// Writes an int64 field value, without a tag, to the stream.
FUNCTION F_WriteInt64 : HRESULT
VAR_INPUT
    stBuffer    : ST_Span;
END_VAR
VAR_IN_OUT
    stState     : ST_WriterInternalState;
END_VAR
VAR_INPUT
    nValue : LINT;
END_VAR
VAR
END_VAR

F_WriteInt64 := F_WriteRawVarint64(stBuffer, stState, nValue);

END_FUNCTION

(* stored: Version 1.1.0.1
   POU F_WriteInt64: Id {2093fb42-8ff6-47d7-b0f8-46c0d2962114}, SpecialFunc None *)
